PROGRAM PRG_Init
VAR_INPUT
	bExecute				: BOOL;		(*Executes initialisation*)
END_VAR
VAR_OUTPUT
	bDone					: BOOL;		(*Initialisation Completed*)
END_VAR
VAR
	fbEnableNetwork_Th1		: FB_EnableNetwork;
	fbEnableNetwork_Th2		: FB_EnableNetwork;
	fbSetVelocityProfile_Th1: FB_SetVelocityProfile;
	fbSetVelocityProfile_Th2: FB_SetVelocityProfile;

	R_DoneTrigger_Th1	: R_TRIG;	(*Bus and controllers has been enabled*)
	R_DoneTrigger_Th2	: R_TRIG;
	
	bSetVeloProfDone		: BOOL := FALSE;
	bStartBusDone			: BOOL := FALSE;
	bBusEnabled				: BOOL;	(*Bus and controllers are enabled*)
END_VAR

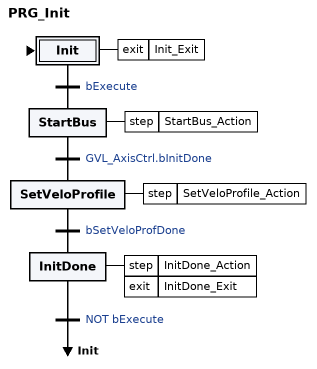
INITIAL_STEP Init:
    Init_Exit(P0);  // exit action
END_STEP
TRANSITION FROM Init TO StartBus
    := bExecute;
END_TRANSITION
STEP StartBus:
    StartBus_Action(N);  // step action
END_STEP
TRANSITION FROM StartBus TO SetVeloProfile
    := GVL_AxisCtrl.bInitDone;
END_TRANSITION
STEP SetVeloProfile:
    SetVeloProfile_Action(N);  // step action
END_STEP
TRANSITION FROM SetVeloProfile TO InitDone
    := bSetVeloProfDone;
END_TRANSITION
STEP InitDone:
    InitDone_Action(N);  // step action
    InitDone_Exit(P0);  // exit action
END_STEP
TRANSITION FROM InitDone TO Init
    := NOT bExecute;
END_TRANSITION

ACTION Init_Exit:
bDone := FALSE;
END_ACTION

ACTION InitDone_Action:
bDone :=TRUE;
END_ACTION

ACTION InitDone_Exit:
bDone :=FALSE;
END_ACTION

ACTION SetVeloProfile:

END_ACTION

ACTION SetVeloProfile_Action:
fbSetVelocityProfile_Th1(
	ADSNetId:= GVL_AxisCtrl.NId ,
	NodeId:=  GVL_AxisCtrl.Th1_NodeAddr,
	Write:= TRUE,
	ProfileAcceleration:= 100000,
	ProfileDeceleration:= 100000,
	Done=> , 
	Err=> , 
	ErrNo=> );
	
fbSetVelocityProfile_Th2(
	ADSNetId:= GVL_AxisCtrl.NId ,
	NodeId:=  GVL_AxisCtrl.Th2_NodeAddr,
	Write:= TRUE,
	ProfileAcceleration:= 100000,
	ProfileDeceleration:= 100000,
	Done=> , 
	Err=> , 
	ErrNo=> );
	
R_DoneTrigger_Th1(CLK:=fbSetVelocityProfile_Th1.Done , Q=> );
R_DoneTrigger_Th2(CLK:=fbSetVelocityProfile_Th2.Done , Q=> );

IF R_DoneTrigger_Th1.Q AND R_DoneTrigger_Th2.Q THEN
	bSetVeloProfDone := TRUE;
END_IF;
END_ACTION

ACTION StartBus_Action:
(*Anabloidaan akselit. Mode: 16#03	= 	ProfileVelocityMode*)
fbEnableNetwork_Th1(
	ADSNetId:= GVL_AxisCtrl.NId,
	NodeId:= GVL_AxisCtrl.Th1_NodeAddr,
	bExcute:= TRUE,
	bEnabled:= TRUE,
	iOpMode:= 16#03,
	bDone=> , 
	bErr=> ,
	iErrNo=> );
	
fbEnableNetwork_Th2(
	ADSNetId:= GVL_AxisCtrl.NId,
	NodeId:= GVL_AxisCtrl.Th2_NodeAddr,
	bExcute:= TRUE,
	bEnabled:= TRUE,
	iOpMode:= 16#03,
	bDone=> , 
	bErr=> ,
	iErrNo=> );
	

R_DoneTrigger_Th1(CLK:=fbEnableNetwork_Th1.bDone , Q=> );
R_DoneTrigger_Th1(CLK:=fbEnableNetwork_Th2.bDone , Q=> );

IF R_DoneTrigger_Th1.Q AND R_DoneTrigger_Th1.Q THEN
	bBusEnabled := TRUE;
	GVL_AxisCtrl.bInitDone := TRUE;
ELSE
	GVL_AxisCtrl.bInitDone := FALSE;
END_IF;

(*Initialisation completed*)
//GVL_AxisCtrl.bInitDone := fbEnableNetwork.bDone;
END_ACTION

END_PROGRAM

(* stored: Version 1.1.0.1, ProductVersion 3.1.4024.2
   POU PRG_Init: Id {4c0774c8-8512-45ec-be0b-121264a5324b}, SpecialFunc None
   Action Init_Exit: Id {cc94ea7d-8da9-4583-a987-dc522219167e}
   Action InitDone_Action: Id {921aaa2a-cf32-44d5-bafb-6faf563228dc}
   Action InitDone_Exit: Id {c18fb484-7e42-4fdc-975c-4de78a5f085a}
   Action SetVeloProfile: Id {71d269e6-6ccc-4930-b2b8-3f198b6a4ea7}
   Action SetVeloProfile_Action: Id {f1bd09bb-a740-4708-bbcf-6e1665ba8461}
   Action StartBus_Action: Id {417888c7-0d13-4d7c-a8b9-f72f69b4ce71} *)
